// TIA Portal V17 export
// export: Created 2023-12-22T15:07:59.8752236Z, ExportSetting WithDefaults, DisplayName Totally Integrated Automation Portal, DisplayVersion V17, DisplayName TIA Portal Openness, DisplayVersion V17, DisplayName TIA Portal Version Control Interface, DisplayVersion V17, DisplayName STEP 7 Professional, DisplayVersion V17, DisplayName STEP 7 Safety, DisplayVersion V17, DisplayName WinCC Advanced, DisplayVersion V17
FUNCTION_BLOCK "Support"   // FB3, LAD
{ S7_Optimized_Access := 'FALSE' }
VERSION : 0.1
// stored: AutoNumber true, IsIECCheckEnabled false, SetENOAutomatically false, UDAEnableTagReadback false
   VAR DB_SPECIFIC
      pipe_in : Array[0..20] of Int;
      pipe_out : Array[0..20] of Int;
      state : Array[0..15] of Bool;
   END_VAR
   VAR CONSTANT
      void : Int;
      "----" : Int := 1;
      "|" : Int := 2;
      "--|--" : Int := 3;
      "--.--" : Int := 4;
      "--|" : Int := 5;
      "--*--" : Int := 6;
      "|--" : Int := 7;
      "↴" : Int := 10;
      "↵" : Int := 11;
      "↳" : Int := 12;
      "↱" : Int := 13;
   END_VAR
   VAR_TEMP   // added for the SCL form of the ladder/FBD networks
      _w1 : Bool;
      _w2 : Bool;
      _w3 : Bool;
      _w4 : Bool;
      _w5 : Bool;
   END_VAR
BEGIN

REGION Network 1: Шаги запуска - заполнение магистрали
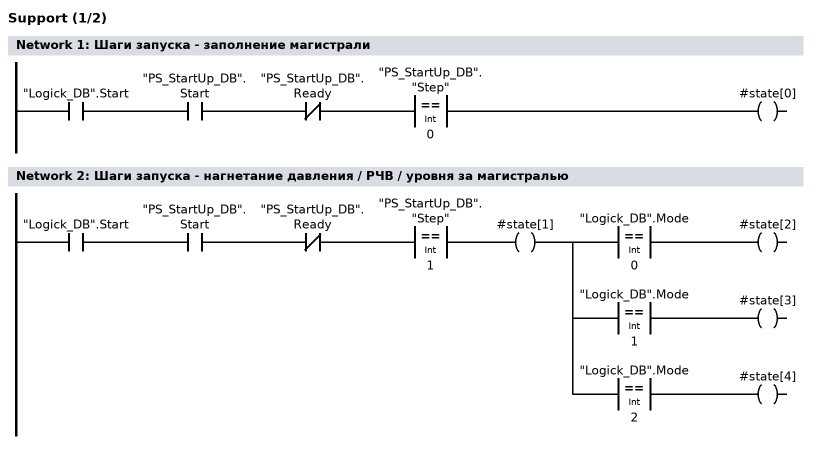
   RUNG wire#powerrail
      Contact( "Logick_DB".Start )
      Contact( "PS_StartUp_DB".Start )
      I_Contact( "PS_StartUp_DB".Ready )
      { S7_Templates := "SrcType := Int" } EQ_Contact(in1 := "PS_StartUp_DB"."Step", in2 := 0)
      Coil( #state[0] )
   END_RUNG
   // the same network as SCL:
   #state[0] := "Logick_DB".Start AND "PS_StartUp_DB".Start AND NOT "PS_StartUp_DB".Ready AND ("PS_StartUp_DB"."Step" = 0);
END_REGION

REGION Network 2: Шаги запуска - нагнетание давления / РЧВ / уровня за магистралью
   RUNG wire#powerrail
      Contact( "Logick_DB".Start )
      Contact( "PS_StartUp_DB".Start )
      I_Contact( "PS_StartUp_DB".Ready )
      { S7_Templates := "SrcType := Int" } EQ_Contact(in1 := "PS_StartUp_DB"."Step", in2 := 1)
      Coil( #state[1] )
      wire#w1
      { S7_Templates := "SrcType := Int" } EQ_Contact(in1 := "Logick_DB".Mode, in2 := 0)
      Coil( #state[2] )
   END_RUNG
   RUNG wire#w1
      { S7_Templates := "SrcType := Int" } EQ_Contact(in1 := "Logick_DB".Mode, in2 := 1)
      Coil( #state[3] )
   END_RUNG
   RUNG wire#w1
      { S7_Templates := "SrcType := Int" } EQ_Contact(in1 := "Logick_DB".Mode, in2 := 2)
      Coil( #state[4] )
   END_RUNG
   // the same network as SCL:
   #state[1] := "Logick_DB".Start AND "PS_StartUp_DB".Start AND NOT "PS_StartUp_DB".Ready AND ("PS_StartUp_DB"."Step" = 1);
   #_w1 := "Logick_DB".Start AND "PS_StartUp_DB".Start AND NOT "PS_StartUp_DB".Ready AND ("PS_StartUp_DB"."Step" = 1);
   #state[2] := #_w1 AND ("Logick_DB".Mode = 0);
   #state[3] := #_w1 AND ("Logick_DB".Mode = 1);
   #state[4] := #_w1 AND ("Logick_DB".Mode = 2);
END_REGION

REGION Network 3: НС-1 - вход
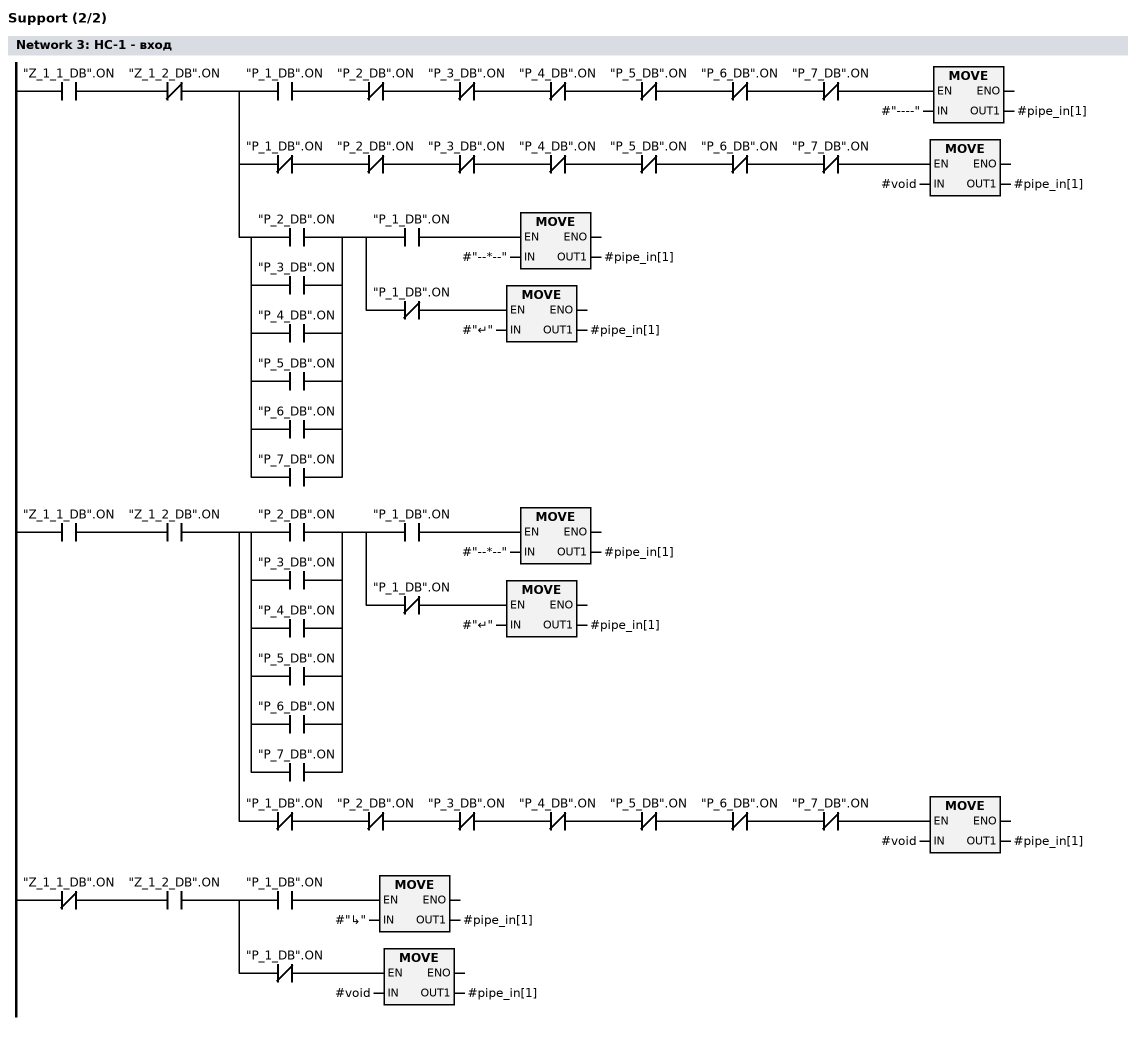
   RUNG wire#powerrail
      Contact( "Z_1_1_DB".ON )
      I_Contact( "Z_1_2_DB".ON )
      wire#w1
      Contact( "P_1_DB".ON )
      I_Contact( "P_2_DB".ON )
      I_Contact( "P_3_DB".ON )
      I_Contact( "P_4_DB".ON )
      I_Contact( "P_5_DB".ON )
      I_Contact( "P_6_DB".ON )
      I_Contact( "P_7_DB".ON )
      Move(in := #"----", out1 => #pipe_in[1])
   END_RUNG
   RUNG wire#w1
      I_Contact( "P_1_DB".ON )
      I_Contact( "P_2_DB".ON )
      I_Contact( "P_3_DB".ON )
      I_Contact( "P_4_DB".ON )
      I_Contact( "P_5_DB".ON )
      I_Contact( "P_6_DB".ON )
      I_Contact( "P_7_DB".ON )
      Move(in := #void, out1 => #pipe_in[1])
   END_RUNG
   RUNG wire#w1
      Contact( "P_2_DB".ON )
      wire#w2
      Contact( "P_1_DB".ON )
      Move(in := #"--*--", out1 => #pipe_in[1])
   END_RUNG
   RUNG wire#w1
      Contact( "P_3_DB".ON )
   END_RUNG wire#w2
   RUNG wire#w1
      Contact( "P_4_DB".ON )
   END_RUNG wire#w2
   RUNG wire#w1
      Contact( "P_5_DB".ON )
   END_RUNG wire#w2
   RUNG wire#w1
      Contact( "P_6_DB".ON )
   END_RUNG wire#w2
   RUNG wire#w1
      Contact( "P_7_DB".ON )
   END_RUNG wire#w2
   RUNG wire#w2
      I_Contact( "P_1_DB".ON )
      Move(in := #"↵", out1 => #pipe_in[1])
   END_RUNG
   RUNG wire#powerrail
      Contact( "Z_1_1_DB".ON )
      Contact( "Z_1_2_DB".ON )
      wire#w3
      Contact( "P_2_DB".ON )
      wire#w4
      Contact( "P_1_DB".ON )
      Move(in := #"--*--", out1 => #pipe_in[1])
   END_RUNG
   RUNG wire#w3
      Contact( "P_3_DB".ON )
   END_RUNG wire#w4
   RUNG wire#w3
      Contact( "P_4_DB".ON )
   END_RUNG wire#w4
   RUNG wire#w3
      Contact( "P_5_DB".ON )
   END_RUNG wire#w4
   RUNG wire#w3
      Contact( "P_6_DB".ON )
   END_RUNG wire#w4
   RUNG wire#w3
      Contact( "P_7_DB".ON )
   END_RUNG wire#w4
   RUNG wire#w4
      I_Contact( "P_1_DB".ON )
      Move(in := #"↵", out1 => #pipe_in[1])
   END_RUNG
   RUNG wire#w3
      I_Contact( "P_1_DB".ON )
      I_Contact( "P_2_DB".ON )
      I_Contact( "P_3_DB".ON )
      I_Contact( "P_4_DB".ON )
      I_Contact( "P_5_DB".ON )
      I_Contact( "P_6_DB".ON )
      I_Contact( "P_7_DB".ON )
      Move(in := #void, out1 => #pipe_in[1])
   END_RUNG
   RUNG wire#powerrail
      I_Contact( "Z_1_1_DB".ON )
      Contact( "Z_1_2_DB".ON )
      wire#w5
      Contact( "P_1_DB".ON )
      Move(in := #"↳", out1 => #pipe_in[1])
   END_RUNG
   RUNG wire#w5
      I_Contact( "P_1_DB".ON )
      Move(in := #void, out1 => #pipe_in[1])
   END_RUNG
   // the same network as SCL:
   #_w1 := "Z_1_1_DB".ON AND NOT "Z_1_2_DB".ON;
   IF #_w1 AND "P_1_DB".ON AND NOT "P_2_DB".ON AND NOT "P_3_DB".ON AND NOT "P_4_DB".ON AND NOT "P_5_DB".ON AND NOT "P_6_DB".ON AND NOT "P_7_DB".ON THEN
       #pipe_in[1] := #"----";
   END_IF;
   IF #_w1 AND NOT "P_1_DB".ON AND NOT "P_2_DB".ON AND NOT "P_3_DB".ON AND NOT "P_4_DB".ON AND NOT "P_5_DB".ON AND NOT "P_6_DB".ON AND NOT "P_7_DB".ON THEN
       #pipe_in[1] := #void;
   END_IF;
   #_w2 := #_w1 AND ("P_2_DB".ON OR "P_3_DB".ON OR "P_4_DB".ON OR "P_5_DB".ON OR "P_6_DB".ON OR "P_7_DB".ON);
   IF #_w2 AND "P_1_DB".ON THEN #pipe_in[1] := #"--*--"; END_IF;
   IF #_w2 AND NOT "P_1_DB".ON THEN #pipe_in[1] := #"↵"; END_IF;
   #_w3 := "Z_1_1_DB".ON AND "Z_1_2_DB".ON;
   #_w4 := #_w3 AND ("P_2_DB".ON OR "P_3_DB".ON OR "P_4_DB".ON OR "P_5_DB".ON OR "P_6_DB".ON OR "P_7_DB".ON);
   IF #_w4 AND "P_1_DB".ON THEN #pipe_in[1] := #"--*--"; END_IF;
   IF #_w4 AND NOT "P_1_DB".ON THEN #pipe_in[1] := #"↵"; END_IF;
   IF #_w3 AND NOT "P_1_DB".ON AND NOT "P_2_DB".ON AND NOT "P_3_DB".ON AND NOT "P_4_DB".ON AND NOT "P_5_DB".ON AND NOT "P_6_DB".ON AND NOT "P_7_DB".ON THEN
       #pipe_in[1] := #void;
   END_IF;
   #_w5 := NOT "Z_1_1_DB".ON AND "Z_1_2_DB".ON;
   IF #_w5 AND "P_1_DB".ON THEN #pipe_in[1] := #"↳"; END_IF;
   IF #_w5 AND NOT "P_1_DB".ON THEN #pipe_in[1] := #void; END_IF;
END_REGION

REGION Network 4: Вентиляция помещений
END_REGION
END_FUNCTION_BLOCK
